/// machine data that is used through most sequences of the unit (motor speed, axes positions, ...)
TYPE MachineDataMachine :
STRUCT
  Slowspeed : LREAL;
  Highspeed : LREAL;
END_STRUCT
END_TYPE

(* stored: Version 1.1.0.1
   DUT MachineDataMachine: Id {5a304f17-0428-4b4b-b0c4-69cf860a1cc2} *)
